// TIA Portal V20 export
DATA_BLOCK "BK10"   // DB205
// stored: MemoryReserve 100
   VAR
      "X10-1 UW TAPE ATTACH V/C ON" : Bool;
      "X10-2 UW TAPE ATTACH V/C OFF" : Bool;
      "X12-1 CART DETECT CHECK LAMP" : Bool;
      "X12-2 SPARE" : Bool;
      "X14-1 SPARE" : Bool;
      "X14-2 SPARE" : Bool;
      "X16-1 SPARE" : Bool;
      "X16-2 SPARE" : Bool;
   END_VAR
BEGIN
END_DATA_BLOCK
